PROGRAM MAIN
VAR
	arr1 : ARRAY [1..100] OF REAL;
	arrayreset : ARRAY [1..100] OF REAL;
	t : ARRAY [1..100]OF REAL;
	i : INT := 1;
	switch : INT := 0;
		
END_VAR


	CASE switch OF
	
		1:
		i := 1;
		t := arrayreset;
		arr1 := arrayreset;
		WHILE i<101 DO
			IF i = 1 
			THEN t[i] := 0.001;
			ELSE t[i] := t[i-1] + 0.001;
			END_IF;
			
			arr1[i] := SIN(t[i]);
			i := i +1;
		END_WHILE
		
		2:
		i := 1;
		t := arrayreset;
		arr1 := arrayreset;
		WHILE i<101 DO
			IF i = 1 
			THEN t[i] := 0.001;
			ELSE t[i] := t[i-1] + 0.001;
			END_IF;
			
			arr1[i] := COS(t[i]);
			i := i +1;
		END_WHILE
		
		3:
		i := 1;
		t := arrayreset;
		arr1 := arrayreset;
		WHILE i<101 DO
			IF i = 1 
			THEN t[i] := 0.001;
			ELSE t[i] := t[i-1] + 0.001;
			END_IF;
			
			arr1[i] := 4* SIN(t[i]);
			i := i +1;
		END_WHILE
		
		
	END_CASE
	//i := 1;
	//t := 0;
	//start := 0;
	//arr1 := arrayreset;

END_PROGRAM

(* stored: Version 1.1.0.1, ProductVersion 3.1.4024.6
   POU MAIN: Id {8e56532f-0f03-40c6-a1a3-b508365bd9a4}, SpecialFunc None *)
